(* PLC project Unnamed, Unknown Unnamed 1 *)
(* stored: creationDateTime 2025-10-10T14:27:24, modificationDateTime 2025-11-03T16:46:36 *)

PROGRAM rd_seq_rbear_trap
  VAR
    START : BOOL;
    PANIC : BOOL;
    Er : BOOL;
    SET_TRAP : BOOL;
    ACTIVATE_TRAP : BOOL;
    IN_MINUTOS : INT := 2;
    IN_SEGUNDOS : INT := 30;
    TIMER : INT;
    C_TIMER : INT;
    D_TIMER : INT;
    DISPLAY_M : INT;
    DISPLAY_S : INT;
    RANDOM : INT;
    RANDOM_ULINT : ULINT;
    SEED : ULINT := 0;
  END_VAR
  VAR CONSTANT
    M10 : ULINT := 10000;
    A : ULINT := 32310901;
    C : ULINT := 32310901;
    M : ULINT := 4294967296;
  END_VAR
  VAR
    Clock : BOOL;
    TOF0 : TOF;
    TON0 : TON;
    CTU_ULINT0 : CTU_ULINT;
    RESET : BOOL;
    D1 : INT;
    D2 : INT;
    D3 : INT;
    D4 : INT;
    CTU0 : CTU;
    R_TRIG1 : R_TRIG;
    CTU1 : CTU;
    TOF1 : TOF;
    CTU2 : CTU;
    TOF2 : TOF;
    CTU3 : CTU;
    TOF3 : TOF;
    CTU4 : CTU;
    TOF4 : TOF;
    B1 : BOOL;
    B2 : BOOL;
    B3 : BOOL;
    B4 : BOOL;
    M1 : BOOL;
    M2 : BOOL;
    M3 : BOOL;
    M4 : BOOL;
    E1 : BOOL;
    E2 : BOOL;
    E3 : BOOL;
    E4 : BOOL;
    R1 : BOOL;
    R2 : BOOL;
    R3 : BOOL;
    R4 : BOOL;
    G0 : BOOL;
    G1 : BOOL;
    G2 : BOOL;
    G3 : BOOL;
    G4 : BOOL;
    O1 : BOOL;
    O2 : BOOL;
    O3 : BOOL;
    O4 : BOOL;
    RELEASE_TRAP : BOOL;
    R_TRIG2 : R_TRIG;
    R_TRIG3 : R_TRIG;
    R_TRIG0 : R_TRIG;
    TON1 : TON;
  END_VAR
  VAR  (* added by the conversion: wires and edge detectors of the diagram *)
    R_TRIG1_2 : R_TRIG;
    R_TRIG2_2 : R_TRIG;
    _MUL1_ENO : BOOL;
    _MUL1_OUT : ULINT;
    _ADD5_ENO : BOOL;
    _ADD5_OUT : ULINT;
    _MOD7_ENO : BOOL;
    _MOD7_OUT : ULINT;
    R_TRIG3_2 : R_TRIG;
    R_TRIG4 : R_TRIG;
    R_TRIG5 : R_TRIG;
    R_TRIG6 : R_TRIG;
    _MUL17_ENO : BOOL;
    _MUL17_OUT : INT;
  END_VAR

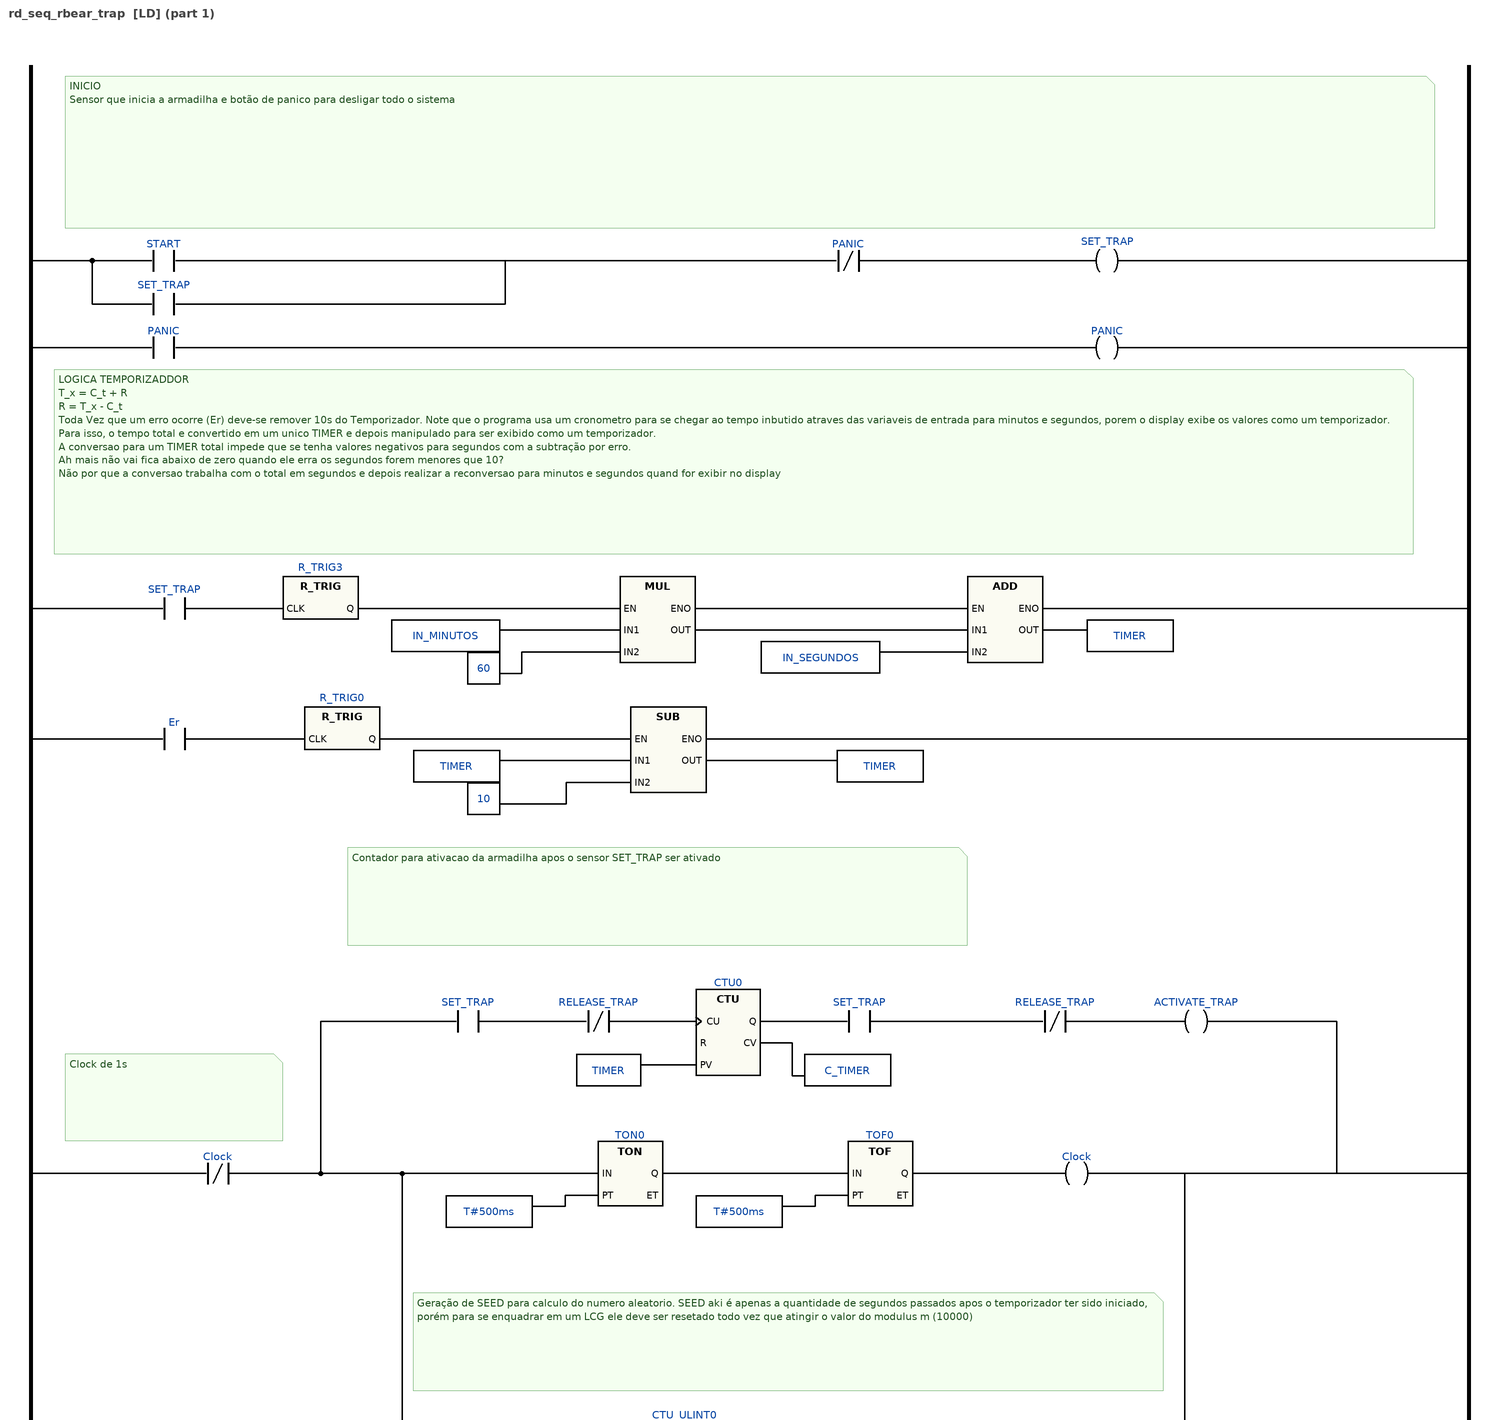
(* LD diagram, written out as Structured Text *)
(* INICIO
Sensor que inicia a armadilha e botão de panico para desligar todo o sistema *)
(* LOGICA TEMPORIZADDOR
T_x = C_t + R
R = T_x - C_t
Toda Vez que um erro ocorre (Er) deve-se remover 10s do Temporizador. Note que o programa usa um cronometro para se chegar ao tempo inbutido atraves das variaveis de entrada para minutos e segundos, porem o display exibe os valores como um temporizador. Para isso, o tempo total e convertido em um unico TIMER e depois manipulado para ser exibido como um temporizador.
A conversao para um TIMER total impede que se tenha valores negativos para segundos com a subtração por erro.
Ah mais não vai fica abaixo de zero quando ele erra os segundos forem menores que 10?
Não por que a conversao trabalha com o total em segundos e depois realizar a reconversao para minutos e segundos quand for exibir no display *)
(* Contador para ativacao da armadilha apos o sensor SET_TRAP ser ativado *)
(* Clock de 1s *)
TON0(IN := NOT Clock, PT := T#500ms);
TOF0(IN := TON0.Q, PT := T#500ms);
Clock := TOF0.Q;
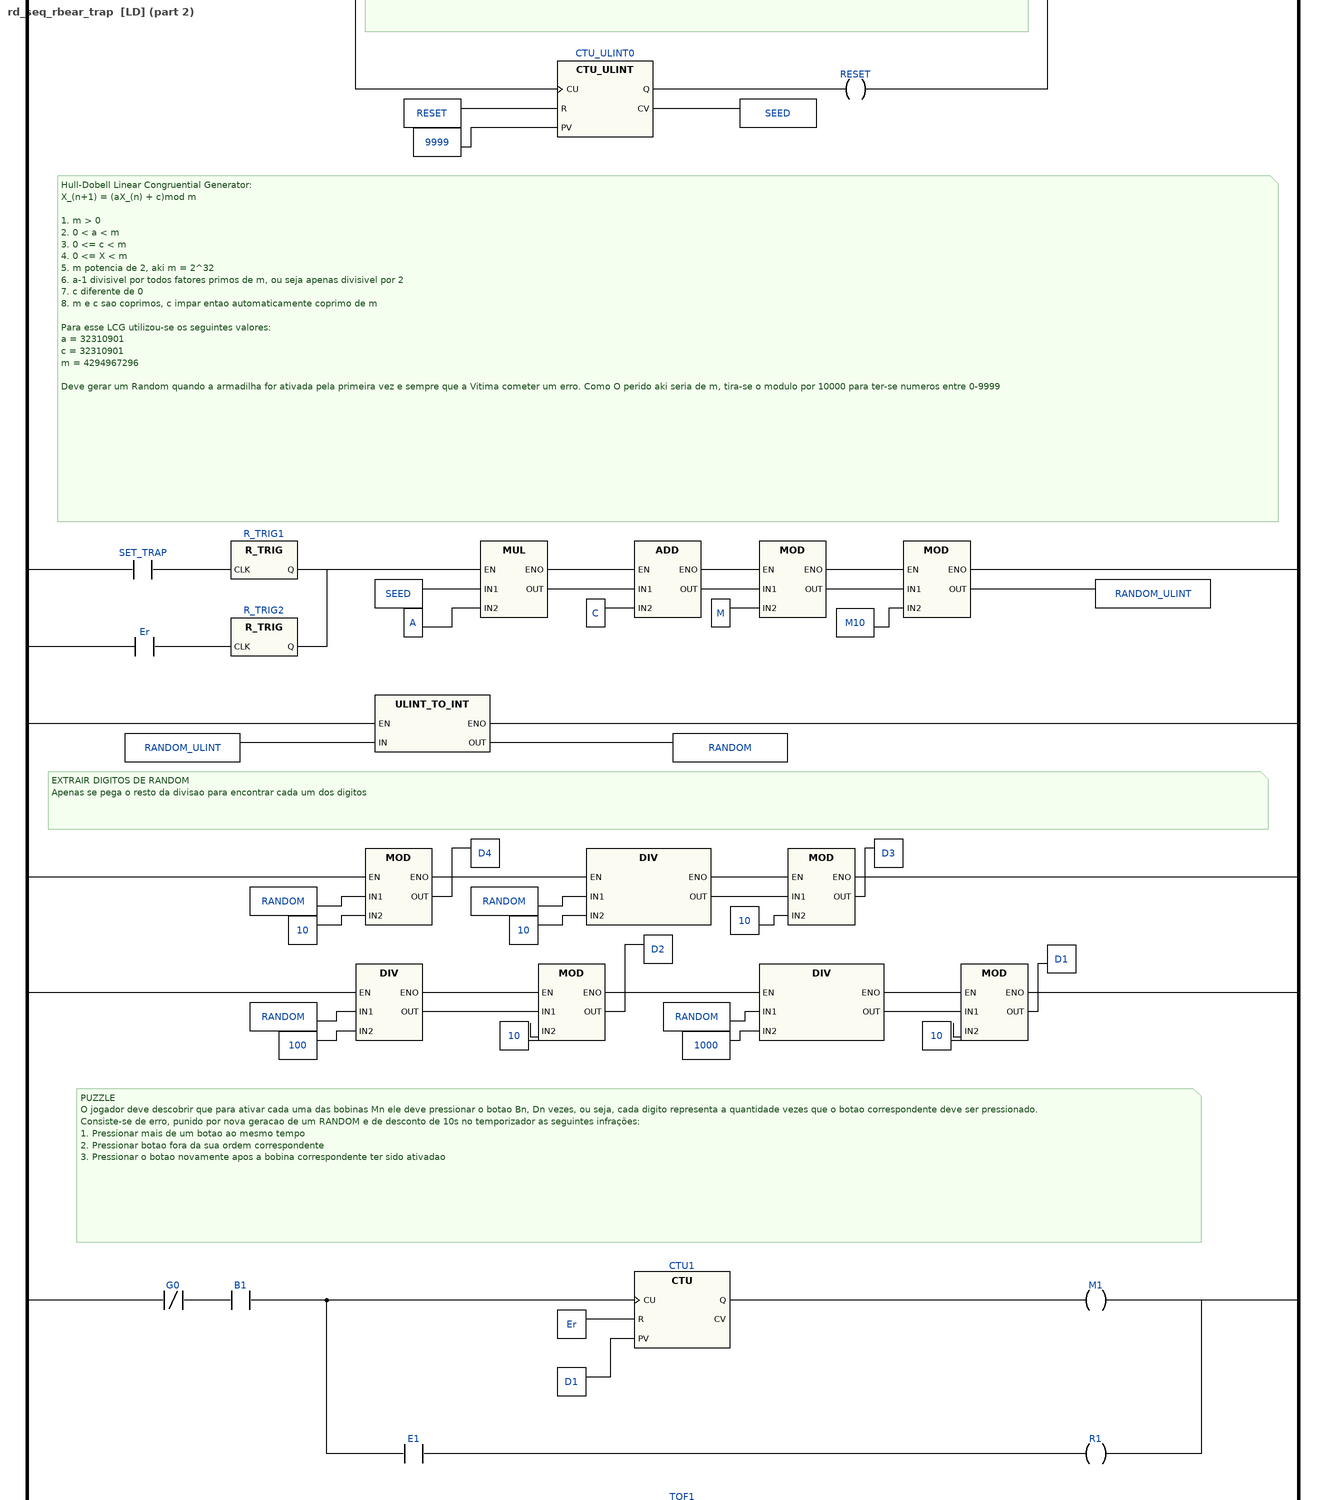
(* Geração de SEED para calculo do numero aleatorio. SEED aki é apenas a quantidade de segundos passados apos o temporizador ter sido iniciado, porém para se enquadrar em um LCG ele deve ser resetado todo vez que atingir o valor do modulus m (10000) *)
R_TRIG1_2(CLK := NOT Clock);
CTU_ULINT0(CU := R_TRIG1_2.Q, R := RESET, PV := 9999);
SEED := CTU_ULINT0.CV;
RESET := CTU_ULINT0.Q;
(* Hull-Dobell Linear Congruential Generator:
X_(n+1) = (aX_(n) + c)mod m

1. m > 0
2. 0 < a < m
3. 0 <= c < m
4. 0 <= X < m
5. m potencia de 2, aki m = 2^32
6. a-1 divisivel por todos fatores primos de m, ou seja apenas divisivel por 2
7. c diferente de 0
8. m e c sao coprimos, c impar entao automaticamente coprimo de m

Para esse LCG utilizou-se os seguintes valores:
   a = 32310901
   c = 32310901
   m = 4294967296

Deve gerar um Random quando a armadilha for ativada pela primeira vez e sempre que a Vitima cometer um erro. Como O perido aki seria de m, tira-se o modulo por 10000 para ter-se numeros entre 0-9999 *)
(* EXTRAIR DIGITOS DE RANDOM
Apenas se pega o resto da divisao para encontrar cada um dos digitos *)
D4 := RANDOM MOD 10;
D3 := RANDOM / 10 MOD 10;
D2 := RANDOM / 100 MOD 10;
D1 := RANDOM / 1000 MOD 10;
R_TRIG2_2(CLK := NOT Clock AND SET_TRAP AND NOT RELEASE_TRAP);
CTU0(CU := R_TRIG2_2.Q, PV := TIMER);
ACTIVATE_TRAP := CTU0.Q AND SET_TRAP AND NOT RELEASE_TRAP;
R_TRIG1(CLK := SET_TRAP);
R_TRIG2(CLK := Er);
_MUL1_OUT := MUL(EN := R_TRIG1.Q OR R_TRIG2.Q, IN1 := SEED, IN2 := A, ENO => _MUL1_ENO);
_ADD5_OUT := ADD(EN := _MUL1_ENO, IN1 := _MUL1_OUT, IN2 := C, ENO => _ADD5_ENO);
_MOD7_OUT := MOD(EN := _ADD5_ENO, IN1 := _ADD5_OUT, IN2 := M, ENO => _MOD7_ENO);
IF _MOD7_ENO THEN RANDOM_ULINT := _MOD7_OUT MOD M10; END_IF;
(* PUZZLE
O jogador deve descobrir que para ativar cada uma das bobinas Mn ele deve pressionar o botao Bn, Dn vezes, ou seja, cada digito representa a quantidade vezes que o botao correspondente deve ser pressionado.
Consiste-se de erro, punido por nova geracao de um RANDOM e de desconto de 10s no temporizador as seguintes infrações:
1. Pressionar mais de um botao ao mesmo tempo
2. Pressionar botao fora da sua ordem correspondente
3. Pressionar o botao novamente apos a bobina correspondente ter sido ativadao *)
R_TRIG3_2(CLK := NOT G0 AND B1);
CTU1(CU := R_TRIG3_2.Q, R := Er, PV := D1);
M1 := CTU1.Q;
R1 := NOT G0 AND B1 AND E1;
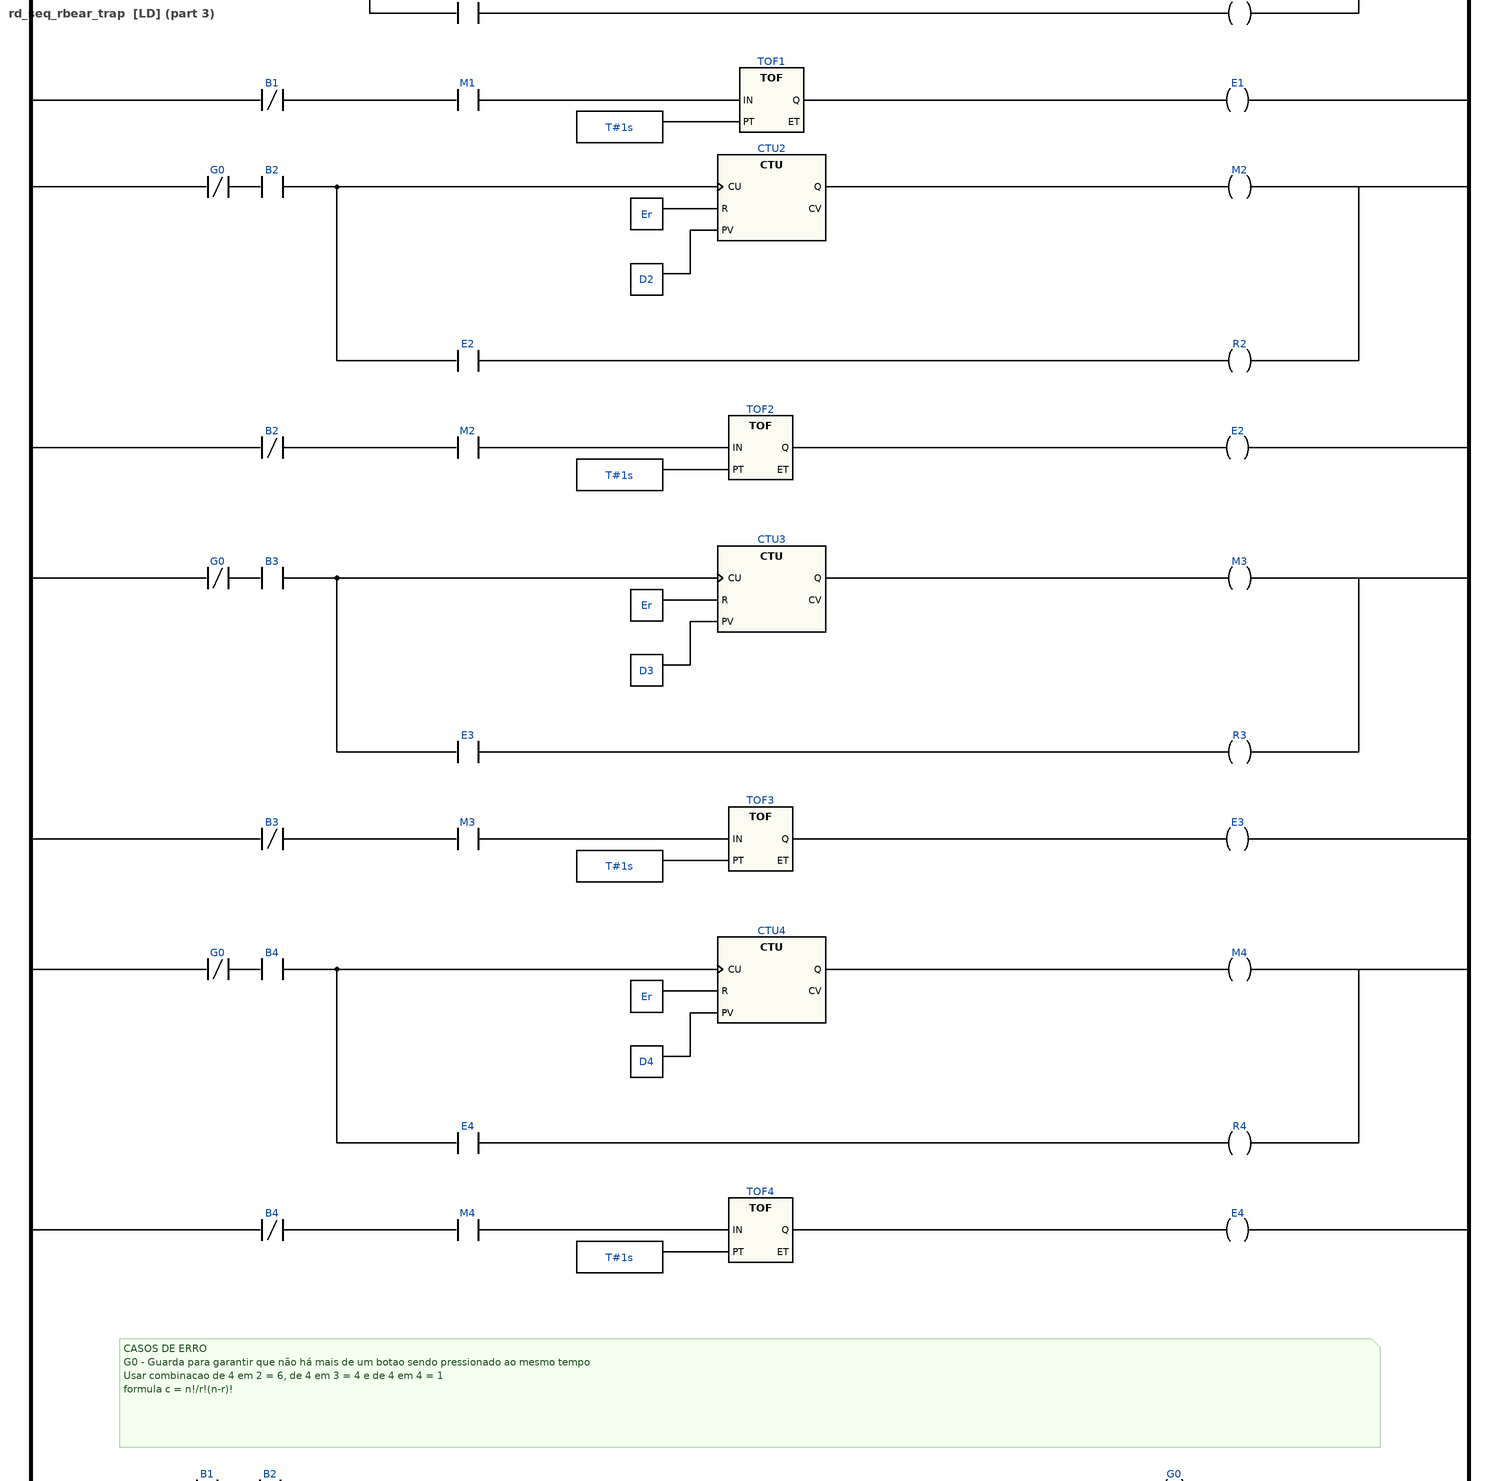
TOF1(IN := NOT B1 AND M1, PT := T#1s);
E1 := TOF1.Q;
R_TRIG4(CLK := NOT G0 AND B2);
CTU2(CU := R_TRIG4.Q, R := Er, PV := D2);
M2 := CTU2.Q;
R2 := NOT G0 AND B2 AND E2;
TOF2(IN := NOT B2 AND M2, PT := T#1s);
E2 := TOF2.Q;
R_TRIG5(CLK := NOT G0 AND B3);
CTU3(CU := R_TRIG5.Q, R := Er, PV := D3);
M3 := CTU3.Q;
R3 := NOT G0 AND B3 AND E3;
TOF3(IN := NOT B3 AND M3, PT := T#1s);
E3 := TOF3.Q;
R_TRIG6(CLK := NOT G0 AND B4);
CTU4(CU := R_TRIG6.Q, R := Er, PV := D4);
M4 := CTU4.Q;
R4 := NOT G0 AND B4 AND E4;
TOF4(IN := NOT B4 AND M4, PT := T#1s);
E4 := TOF4.Q;
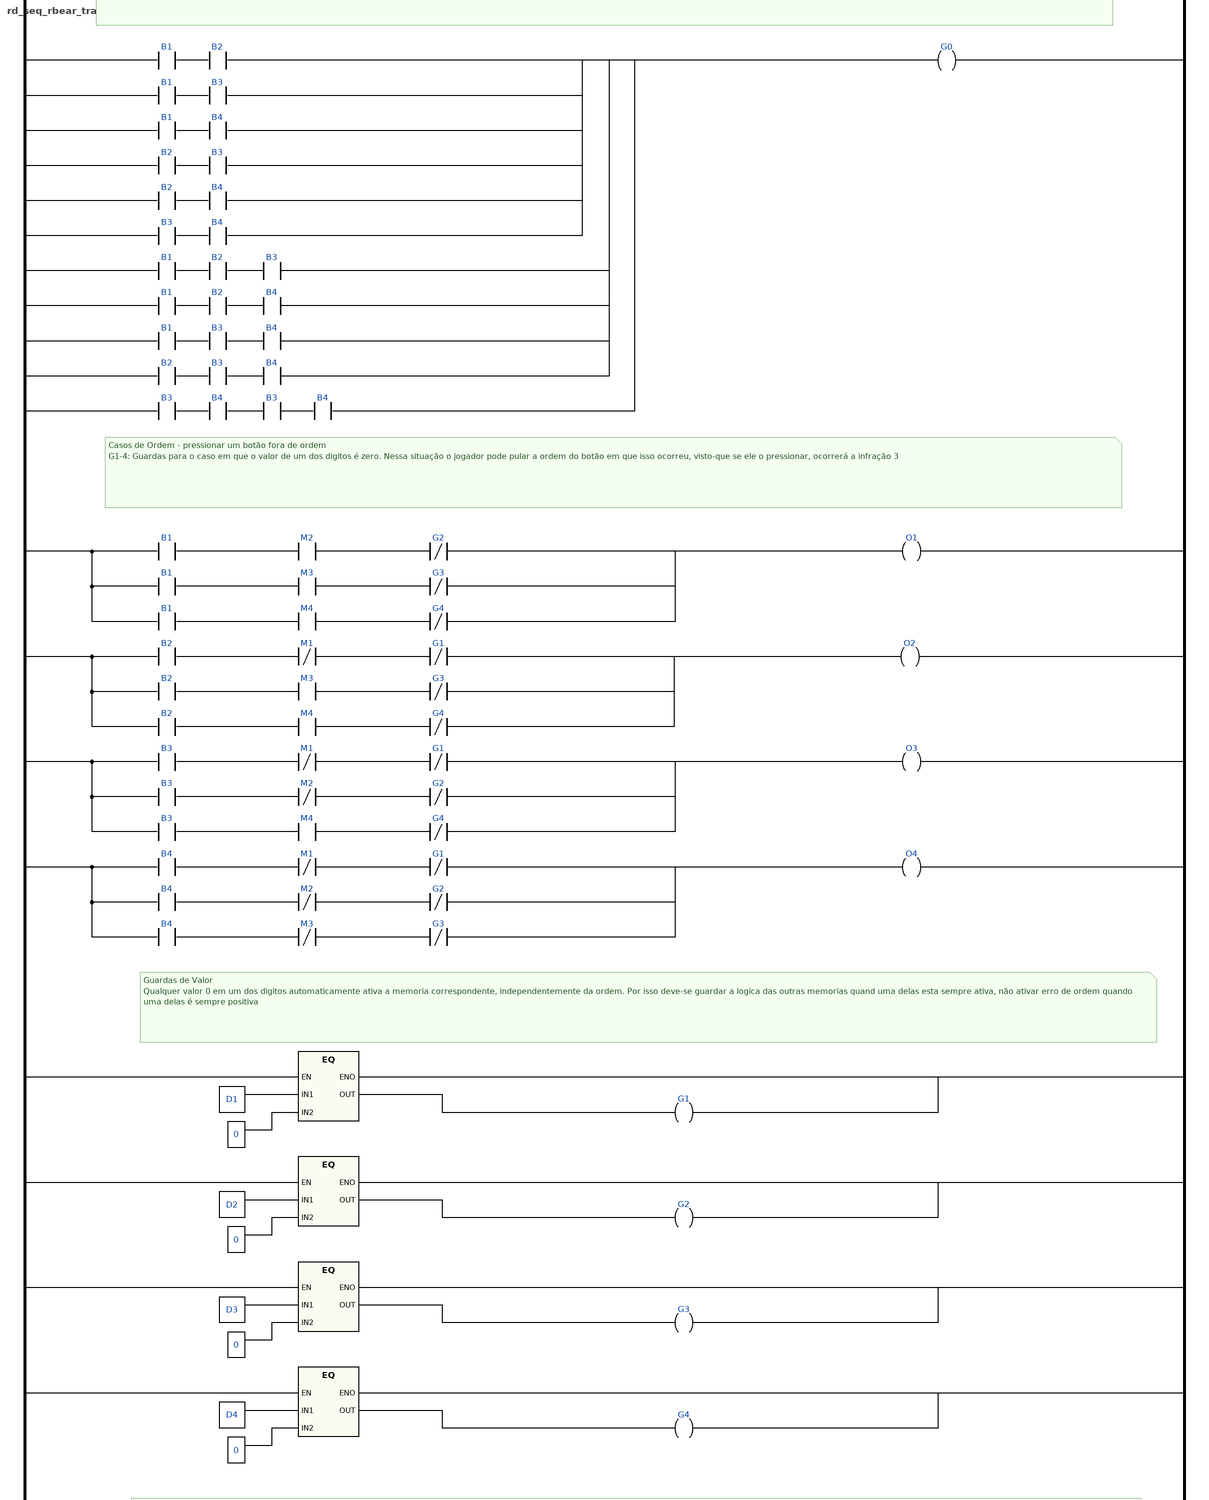
(* CASOS DE ERRO
G0 - Guarda para garantir que não há mais de um botao sendo pressionado ao mesmo tempo
Usar combinacao de 4 em 2 = 6, de 4 em 3 = 4 e de 4 em 4 = 1 
formula c = n!/r!(n-r)! *)
G0 := B1 AND B2 OR B1 AND B3 OR B1 AND B4 OR B2 AND B3 OR B2 AND B4 OR B3 AND B4 OR B1 AND B2 AND B3 OR B1 AND B2 AND B4 OR B1 AND B3 AND B4 OR B2 AND B3 AND B4 OR B3 AND B4 AND B3 AND B4;
(* Casos de Ordem - pressionar um botão fora de ordem
G1-4: Guardas para o caso em que o valor de um dos digitos é zero. Nessa situação o jogador pode pular a ordem do botão em que isso ocorreu, visto-que se ele o pressionar, ocorrerá a infração 3 *)
O1 := B1 AND (M2 AND NOT G2 OR M3 AND NOT G3 OR M4 AND NOT G4);
O2 := B2 AND (NOT M1 AND NOT G1 OR M3 AND NOT G3 OR M4 AND NOT G4);
O3 := B3 AND (NOT M1 AND NOT G1 OR NOT M2 AND NOT G2 OR M4 AND NOT G4);
O4 := B4 AND (NOT M1 AND NOT G1 OR NOT M2 AND NOT G2 OR NOT M3 AND NOT G3);
(* Guardas de Valor
Qualquer valor 0 em um dos digitos automaticamente ativa a memoria correspondente, independentemente da ordem. Por isso deve-se guardar a logica das outras memorias quand uma delas esta sempre ativa, não ativar erro de ordem quando uma delas é sempre positiva *)
G1 := D1 = 0;
G2 := D2 = 0;
G3 := D3 = 0;
G4 := D4 = 0;
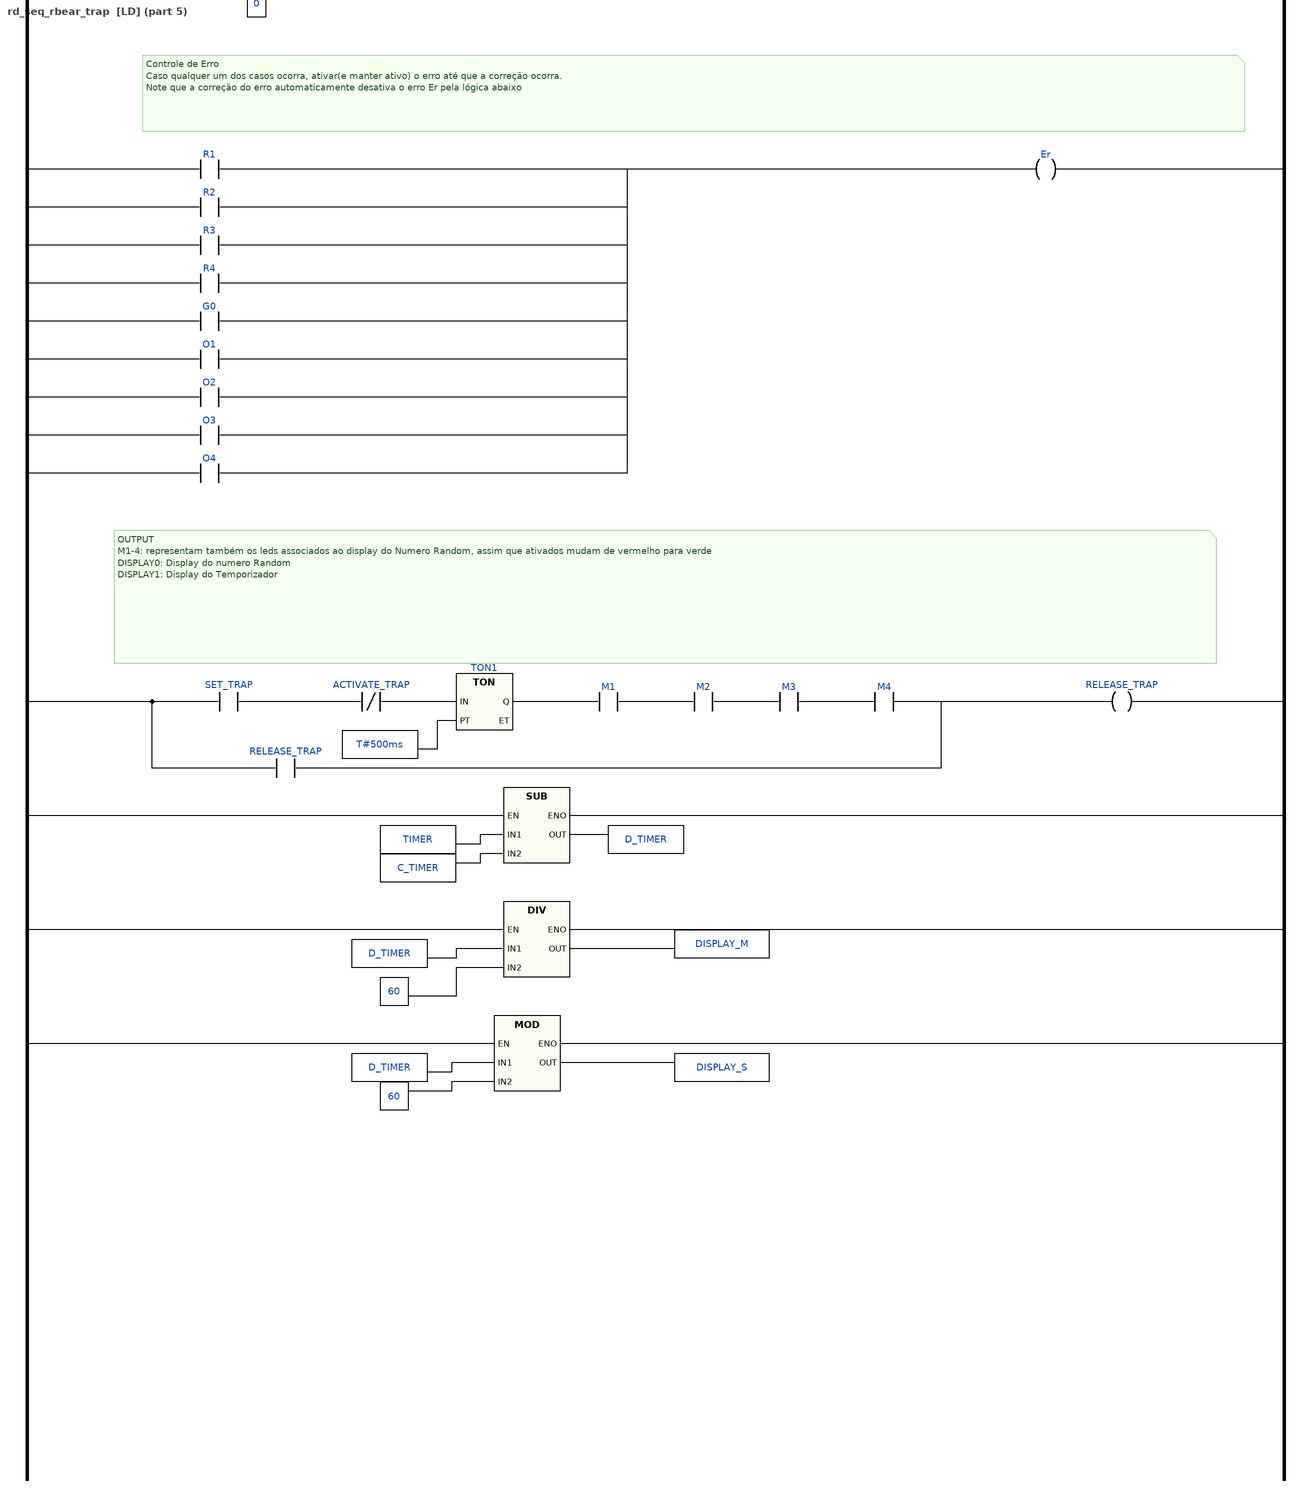
(* Controle de Erro
Caso qualquer um dos casos ocorra, ativar(e manter ativo) o erro até que a correção ocorra.
Note que a correção do erro automaticamente desativa o erro Er pela lógica abaixo *)
Er := R1 OR R2 OR R3 OR R4 OR G0 OR O1 OR O2 OR O3 OR O4;
(* OUTPUT
M1-4: representam também os leds associados ao display do Numero Random, assim que ativados mudam de vermelho para verde
DISPLAY0: Display do numero Random
DISPLAY1: Display do Temporizador *)
TON1(IN := SET_TRAP AND NOT ACTIVATE_TRAP, PT := T#500ms);
RELEASE_TRAP := TON1.Q AND M1 AND M2 AND M3 AND M4 OR RELEASE_TRAP;
RANDOM := ULINT_TO_INT(RANDOM_ULINT);
SET_TRAP := (START OR SET_TRAP) AND NOT PANIC;
PANIC := PANIC;
R_TRIG3(CLK := SET_TRAP);
_MUL17_OUT := MUL(EN := R_TRIG3.Q, IN1 := IN_MINUTOS, IN2 := 60, ENO => _MUL17_ENO);
IF _MUL17_ENO THEN TIMER := _MUL17_OUT + IN_SEGUNDOS; END_IF;
R_TRIG0(CLK := Er);
IF R_TRIG0.Q THEN TIMER := TIMER - 10; END_IF;
C_TIMER := CTU0.CV;
DISPLAY_S := D_TIMER MOD 60;
DISPLAY_M := D_TIMER / 60;
D_TIMER := TIMER - C_TIMER;
END_PROGRAM

PROGRAM my_clock_counter
  VAR
    Clock : BOOL;
    Clock0 : BOOL;
    DISPLAY : ULINT;
    TON0 : TON;
    TOF0 : TOF;
    CTU_ULINT0 : CTU_ULINT;
    Reset : BOOL;
  END_VAR
  VAR  (* added by the conversion: wires and edge detectors of the diagram *)
    R_TRIG1 : R_TRIG;
  END_VAR

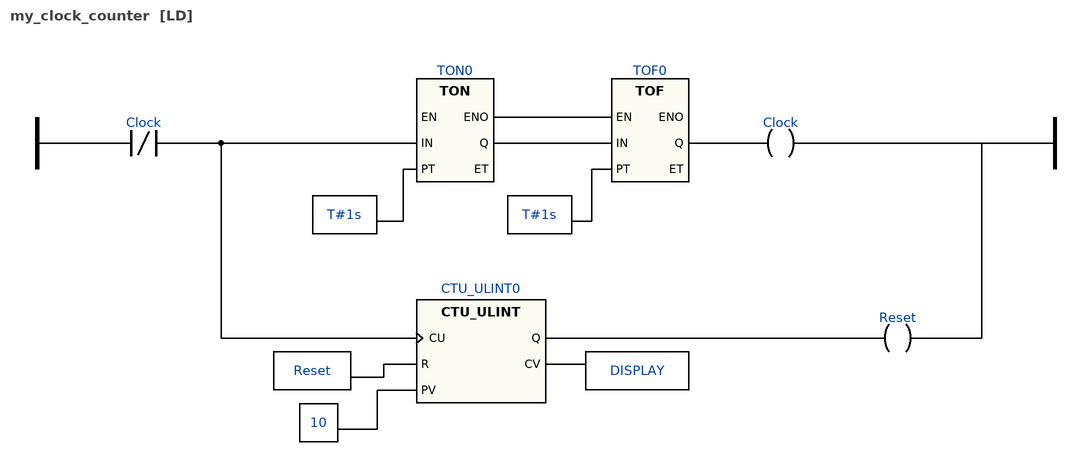
(* LD diagram, written out as Structured Text *)
TON0(IN := NOT Clock, PT := T#1s);
TOF0(EN := TON0.ENO, IN := TON0.Q, PT := T#1s);
Clock := TOF0.Q;
R_TRIG1(CLK := NOT Clock);
CTU_ULINT0(CU := R_TRIG1.Q, R := Reset, PV := 10);
DISPLAY := CTU_ULINT0.CV;
Reset := CTU_ULINT0.Q;
END_PROGRAM

PROGRAM digit_extractor
  VAR
    RANDOM : ULINT := 1234;
    DIVISOR : ULINT := 10;
  END_VAR
  VAR RETAIN
    D1 : ULINT;
  END_VAR
  VAR
    D2 : ULINT;
    D3 : ULINT;
    D4 : ULINT;
    M1 : BOOL;
  END_VAR

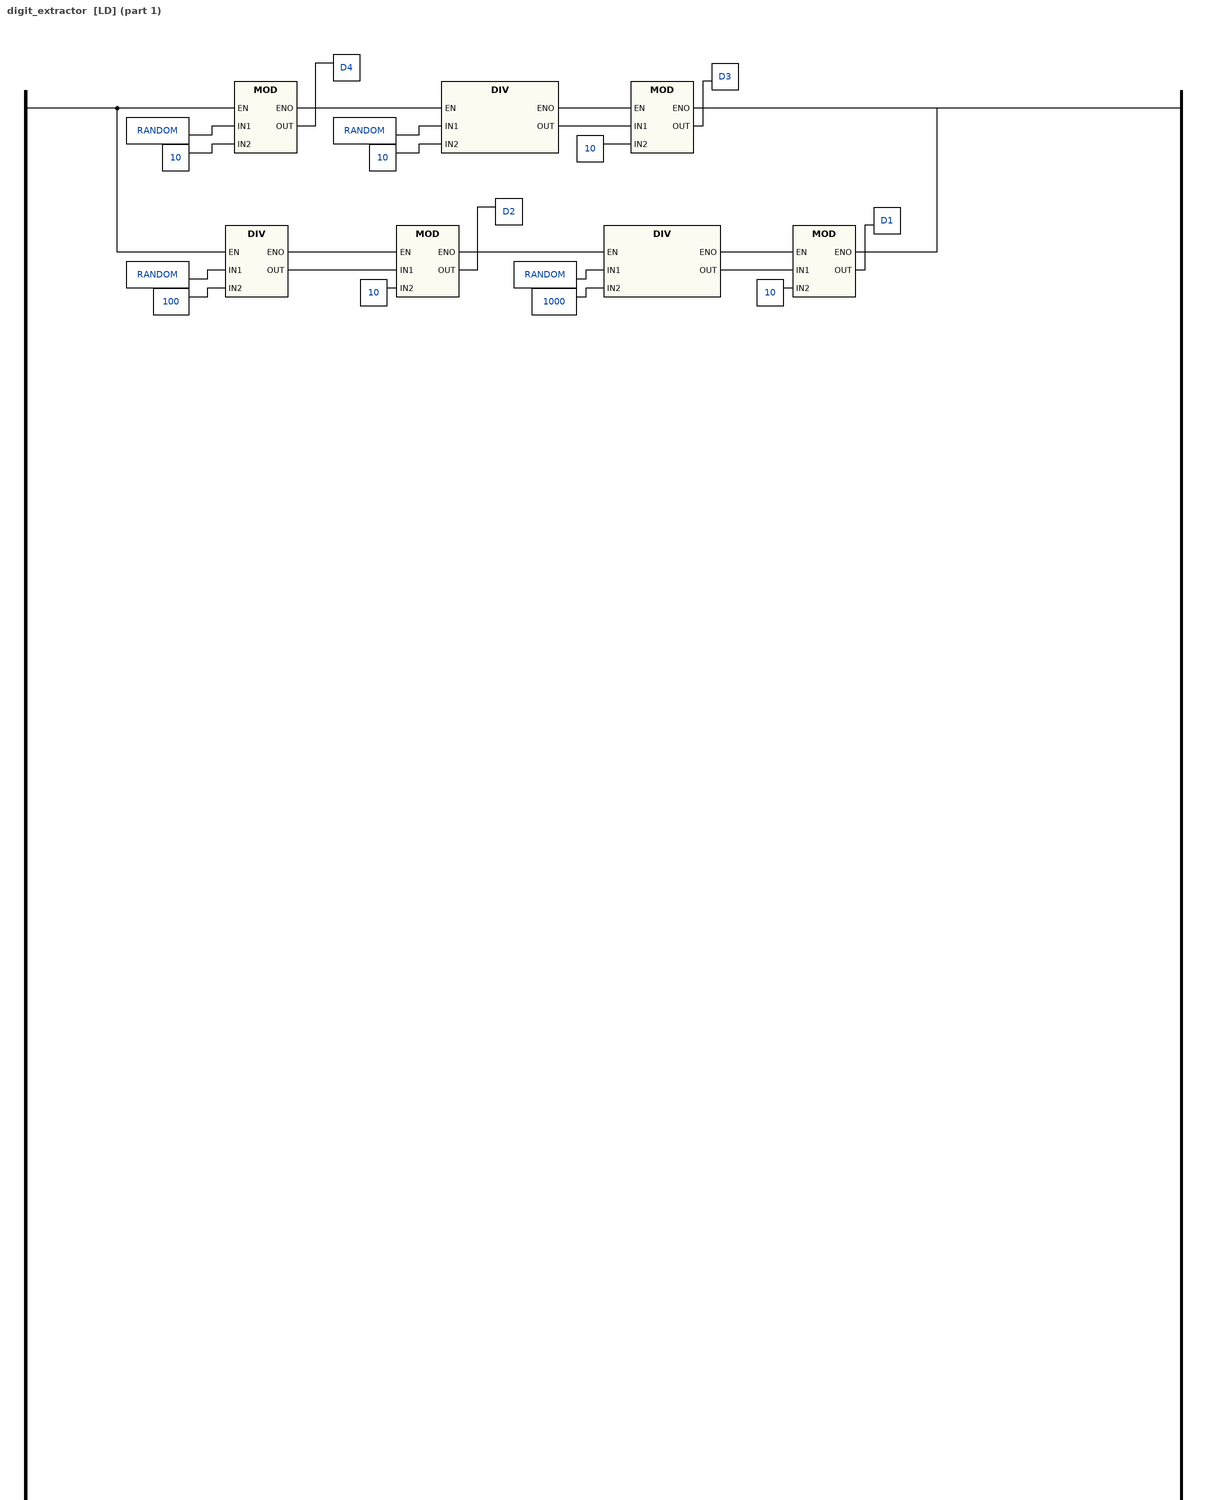
(* LD diagram, written out as Structured Text *)
D4 := RANDOM MOD 10;
D3 := RANDOM / 10 MOD 10;
D2 := RANDOM / 100 MOD 10;
D1 := RANDOM / 1000 MOD 10;
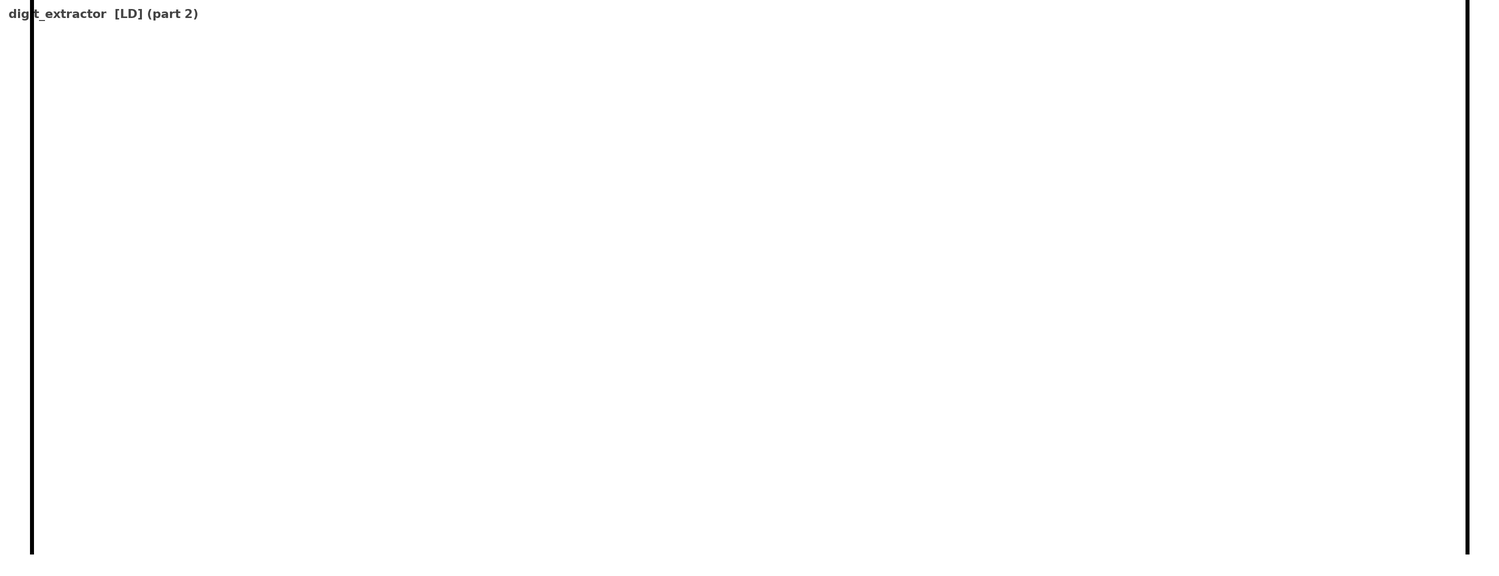
END_PROGRAM

PROGRAM puzzle
  VAR
    D1 : INT := 1;
    D2 : INT := 1;
    D3 : INT := 1;
    D4 : INT := 1;
    B1 : BOOL;
    B2 : BOOL;
    B3 : BOOL;
    B4 : BOOL;
    M1 : BOOL;
    M2 : BOOL;
    M3 : BOOL;
    M4 : BOOL;
    E1 : BOOL;
    E2 : BOOL;
    E3 : BOOL;
    E4 : BOOL;
    CTU1 : CTU;
    R1 : BOOL;
    R2 : BOOL;
    R3 : BOOL;
    R4 : BOOL;
    G1 : BOOL;
    G2 : BOOL;
    G3 : BOOL;
    G4 : BOOL;
    G0 : BOOL;
    O1 : BOOL;
    O2 : BOOL;
    O3 : BOOL;
    O4 : BOOL;
    Er : BOOL;
    SAFE : BOOL;
    CTU2 : CTU;
    CTU3 : CTU;
    CTU4 : CTU;
  END_VAR
  VAR  (* added by the conversion: wires and edge detectors of the diagram *)
    R_TRIG1 : R_TRIG;
    R_TRIG2 : R_TRIG;
    R_TRIG3 : R_TRIG;
    R_TRIG4 : R_TRIG;
  END_VAR

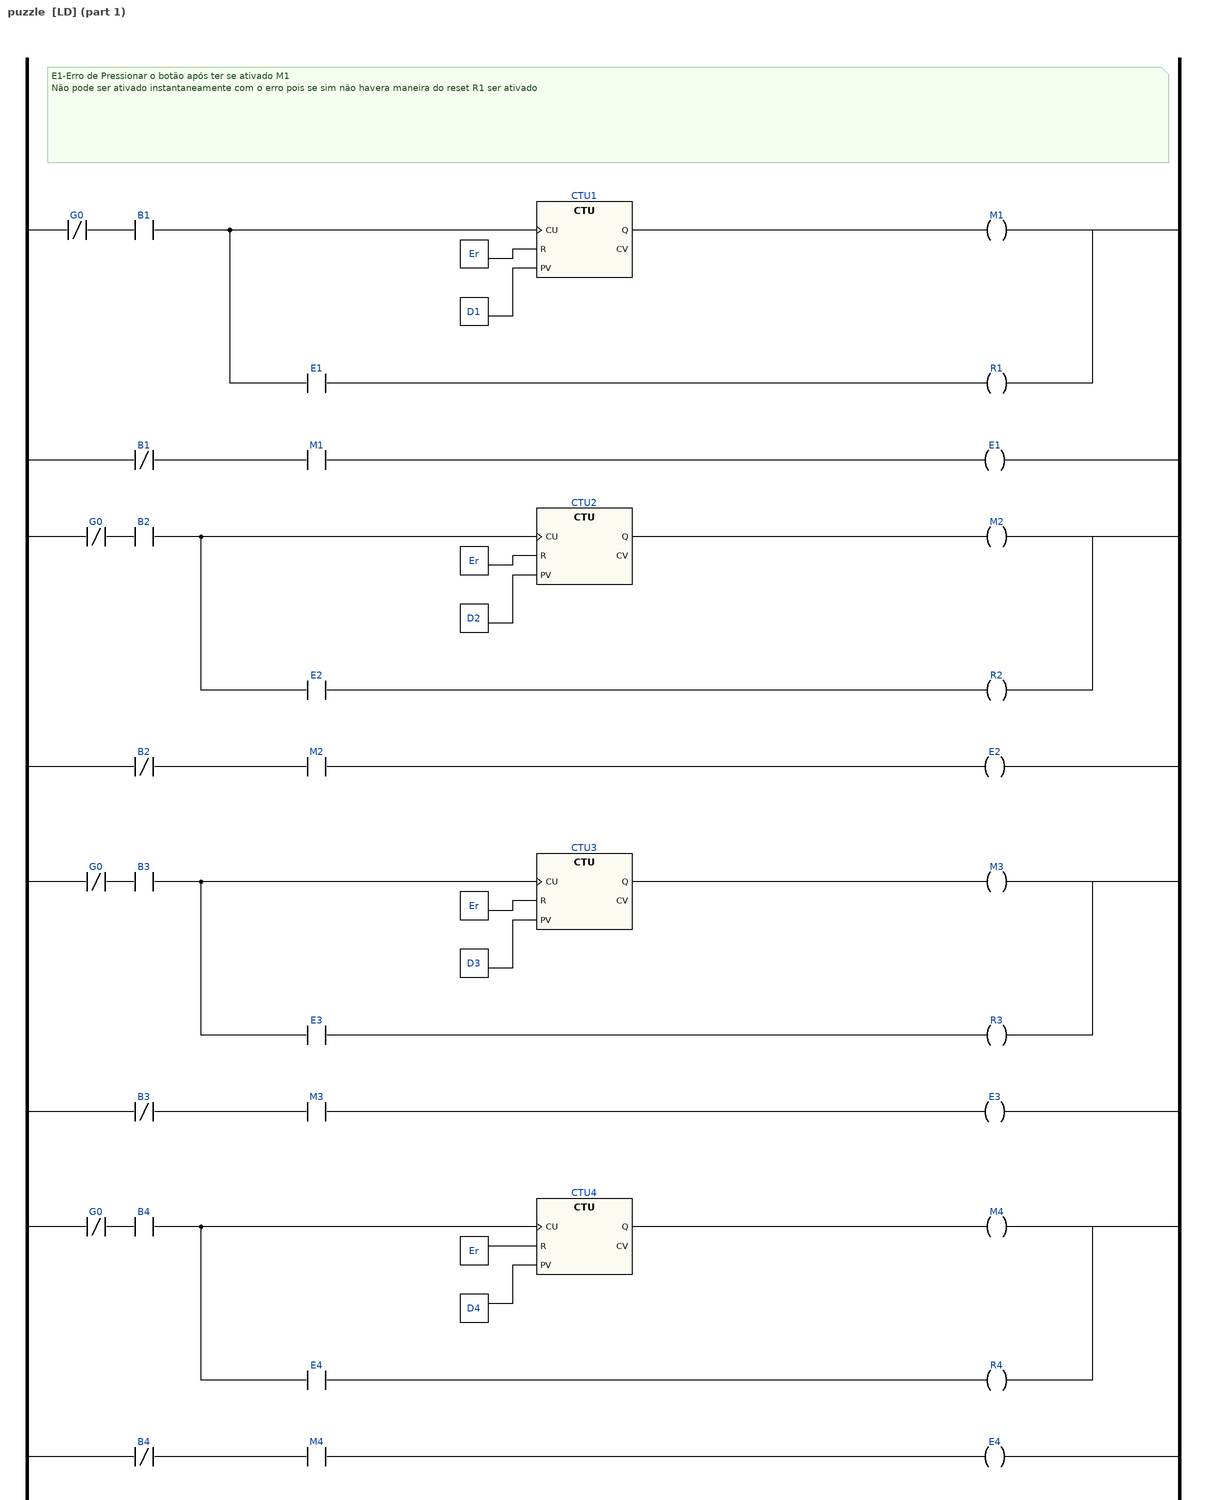
(* LD diagram, written out as Structured Text *)
(* E1-Erro de Pressionar o botão após ter se ativado M1
Não pode ser ativado instantaneamente com o erro pois se sim não havera maneira do reset R1 ser ativado *)
R_TRIG1(CLK := NOT G0 AND B1);
CTU1(CU := R_TRIG1.Q, R := Er, PV := D1);
M1 := CTU1.Q;
R1 := NOT G0 AND B1 AND E1;
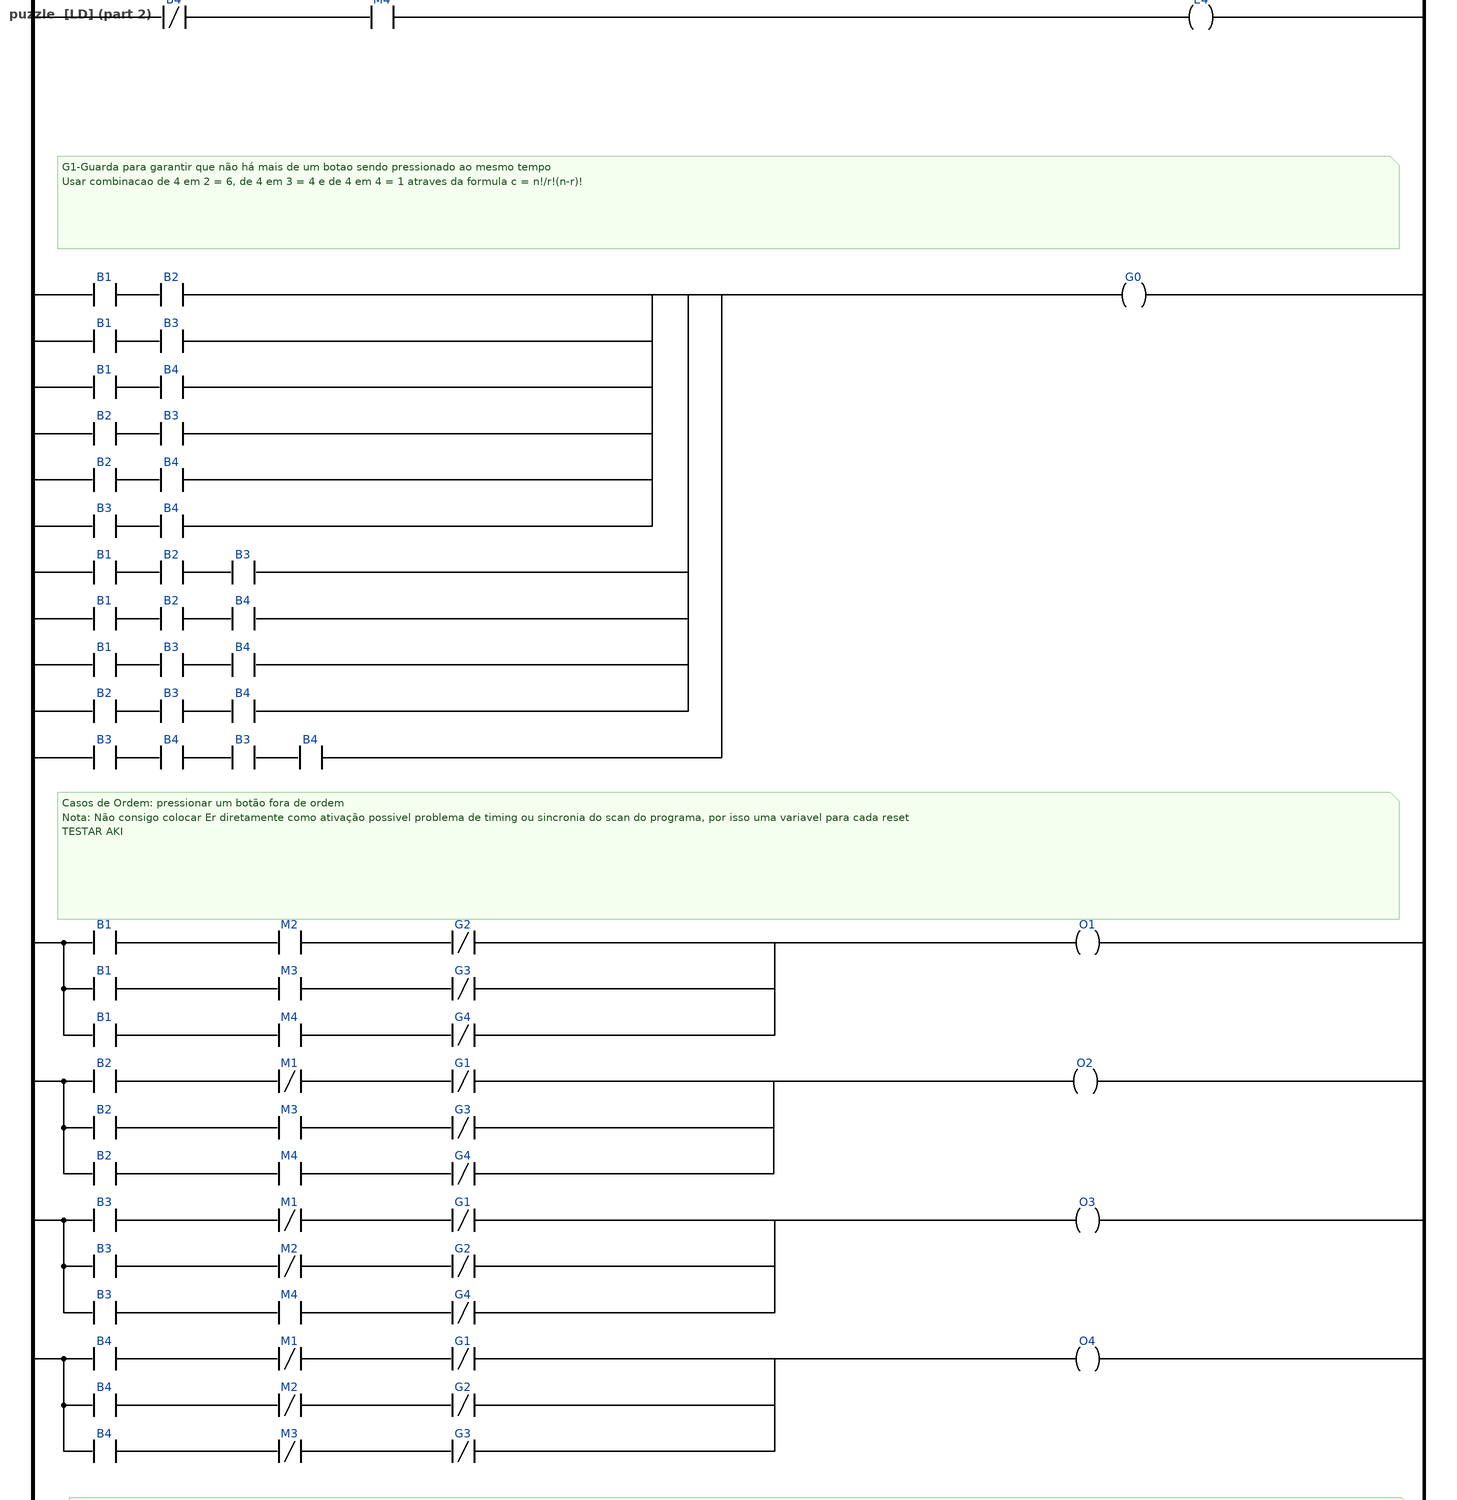
(* G1-Guarda para garantir que não há mais de um botao sendo pressionado ao mesmo tempo
Usar combinacao de 4 em 2 = 6, de 4 em 3 = 4 e de 4 em 4 = 1 atraves da formula c = n!/r!(n-r)! *)
G0 := B1 AND B2 OR B1 AND B3 OR B1 AND B4 OR B2 AND B3 OR B2 AND B4 OR B3 AND B4 OR B1 AND B2 AND B3 OR B1 AND B2 AND B4 OR B1 AND B3 AND B4 OR B2 AND B3 AND B4 OR B3 AND B4 AND B3 AND B4;
(* Casos de Ordem: pressionar um botão fora de ordem
Nota: Não consigo colocar Er diretamente como ativação possivel problema de timing ou sincronia do scan do programa, por isso uma variavel para cada reset
TESTAR AKI *)
O1 := B1 AND (M2 AND NOT G2 OR M3 AND NOT G3 OR M4 AND NOT G4);
R_TRIG2(CLK := NOT G0 AND B2);
CTU2(CU := R_TRIG2.Q, R := Er, PV := D2);
M2 := CTU2.Q;
R2 := NOT G0 AND B2 AND E2;
E2 := NOT B2 AND M2;
R_TRIG3(CLK := NOT G0 AND B3);
CTU3(CU := R_TRIG3.Q, R := Er, PV := D3);
M3 := CTU3.Q;
R3 := NOT G0 AND B3 AND E3;
E3 := NOT B3 AND M3;
R_TRIG4(CLK := NOT G0 AND B4);
CTU4(CU := R_TRIG4.Q, R := Er, PV := D4);
M4 := CTU4.Q;
R4 := NOT G0 AND B4 AND E4;
E4 := NOT B4 AND M4;
O2 := B2 AND (NOT M1 AND NOT G1 OR M3 AND NOT G3 OR M4 AND NOT G4);
O3 := B3 AND (NOT M1 AND NOT G1 OR NOT M2 AND NOT G2 OR M4 AND NOT G4);
O4 := B4 AND (NOT M1 AND NOT G1 OR NOT M2 AND NOT G2 OR NOT M3 AND NOT G3);
E1 := NOT B1 AND M1;
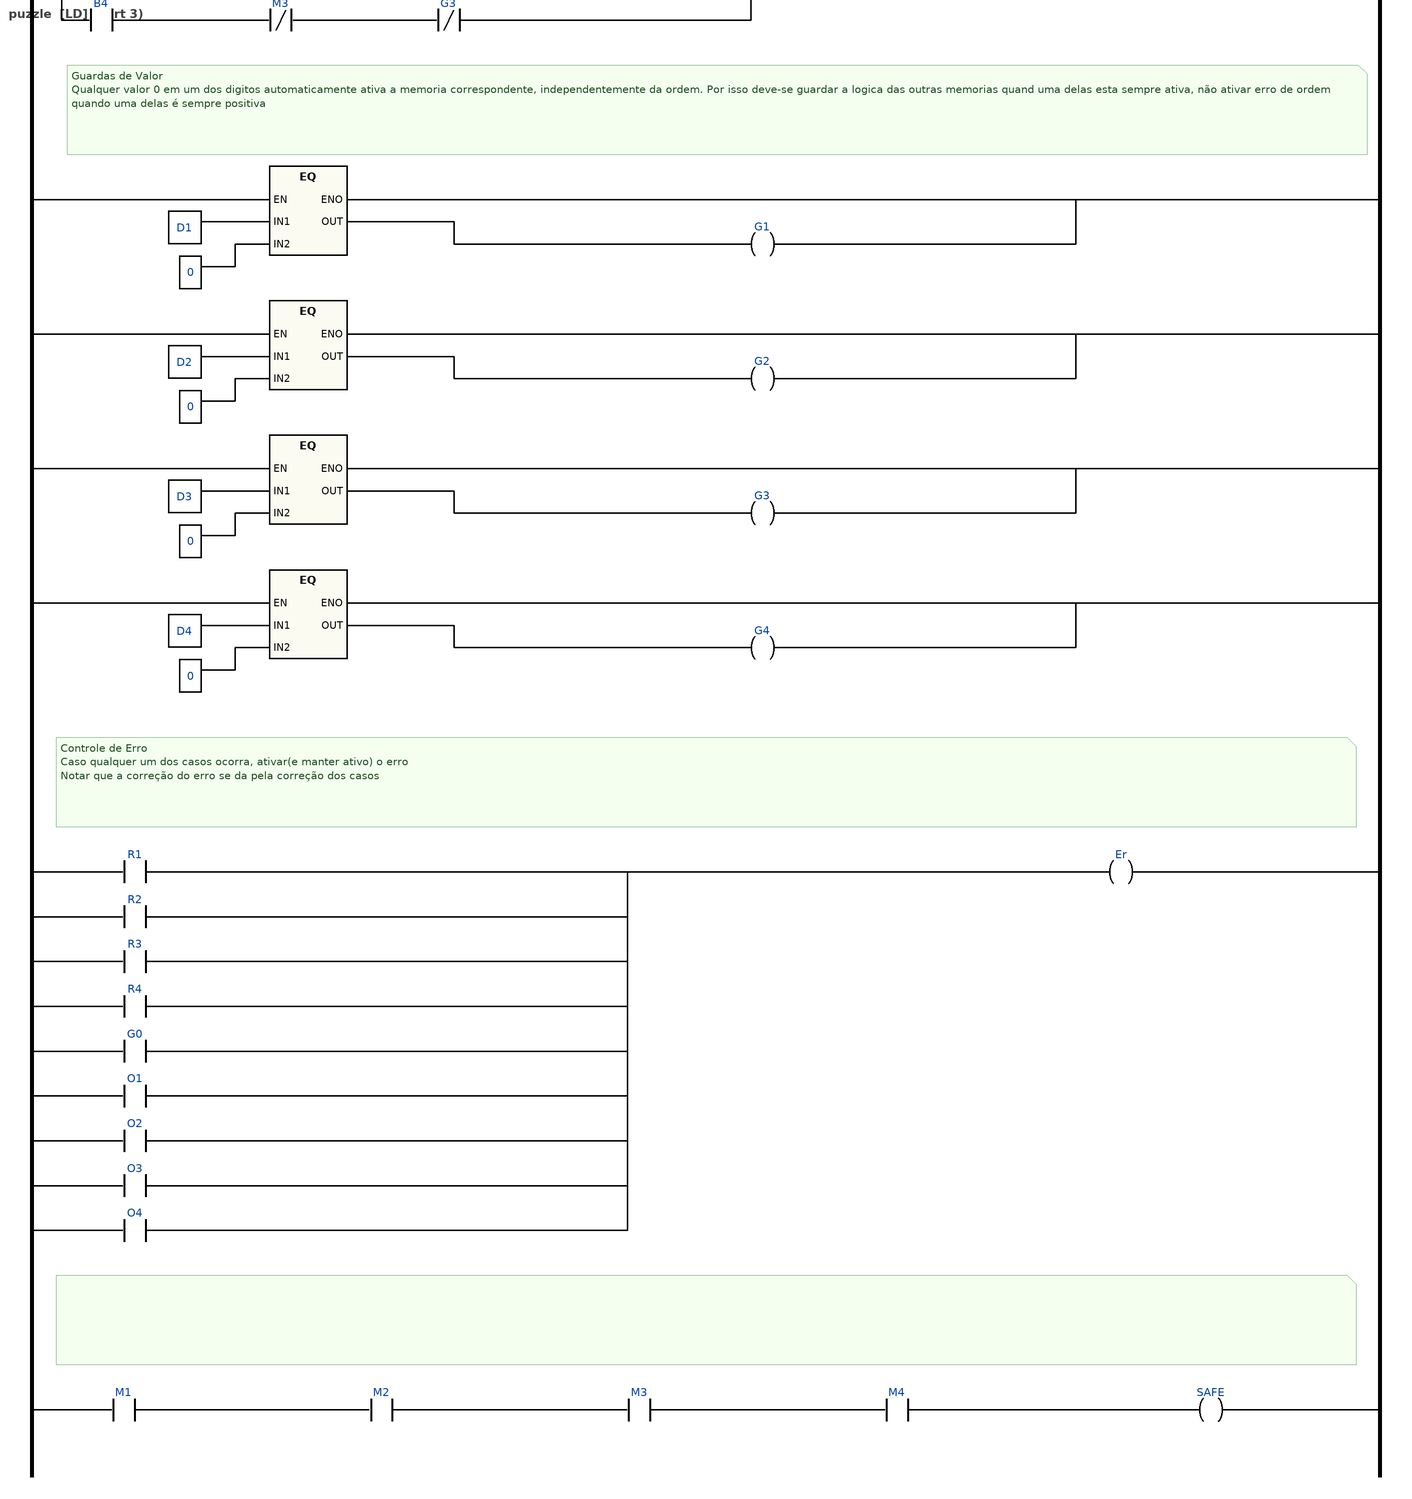
(* Guardas de Valor
Qualquer valor 0 em um dos digitos automaticamente ativa a memoria correspondente, independentemente da ordem. Por isso deve-se guardar a logica das outras memorias quand uma delas esta sempre ativa, não ativar erro de ordem quando uma delas é sempre positiva *)
G1 := D1 = 0;
G2 := D2 = 0;
G3 := D3 = 0;
G4 := D4 = 0;
(* Controle de Erro
Caso qualquer um dos casos ocorra, ativar(e manter ativo) o erro
Notar que a correção do erro se da pela correção dos casos *)
Er := R1 OR R2 OR R3 OR R4 OR G0 OR O1 OR O2 OR O3 OR O4;
SAFE := M1 AND M2 AND M3 AND M4;
END_PROGRAM

PROGRAM sub_timer
  VAR
    Er : BOOL;
    START : BOOL;
    PANIC : BOOL;
    IN_MINUTOS : INT := 2;
    IN_SEGUNDOS : INT := 20;
    R_SEGUNDOS : BOOL;
    DISPLAY_M : INT;
    DISPLAY_S : INT;
    Clock : BOOL;
    I_TIMER : INT;
    TIMER : INT;
    C_TIMER : INT;
    D_TIMER : INT;
    TOF0 : TOF;
    TON0 : TON;
    SET_TRAP : BOOL;
    ACTIVATE_TRAP : BOOL;
    CTU0 : CTU;
    R_TRIG0 : R_TRIG;
    R_TRIG1 : R_TRIG;
  END_VAR
  VAR  (* added by the conversion: wires and edge detectors of the diagram *)
    R_TRIG1_2 : R_TRIG;
    _MUL86_ENO : BOOL;
    _MUL86_OUT : INT;
  END_VAR

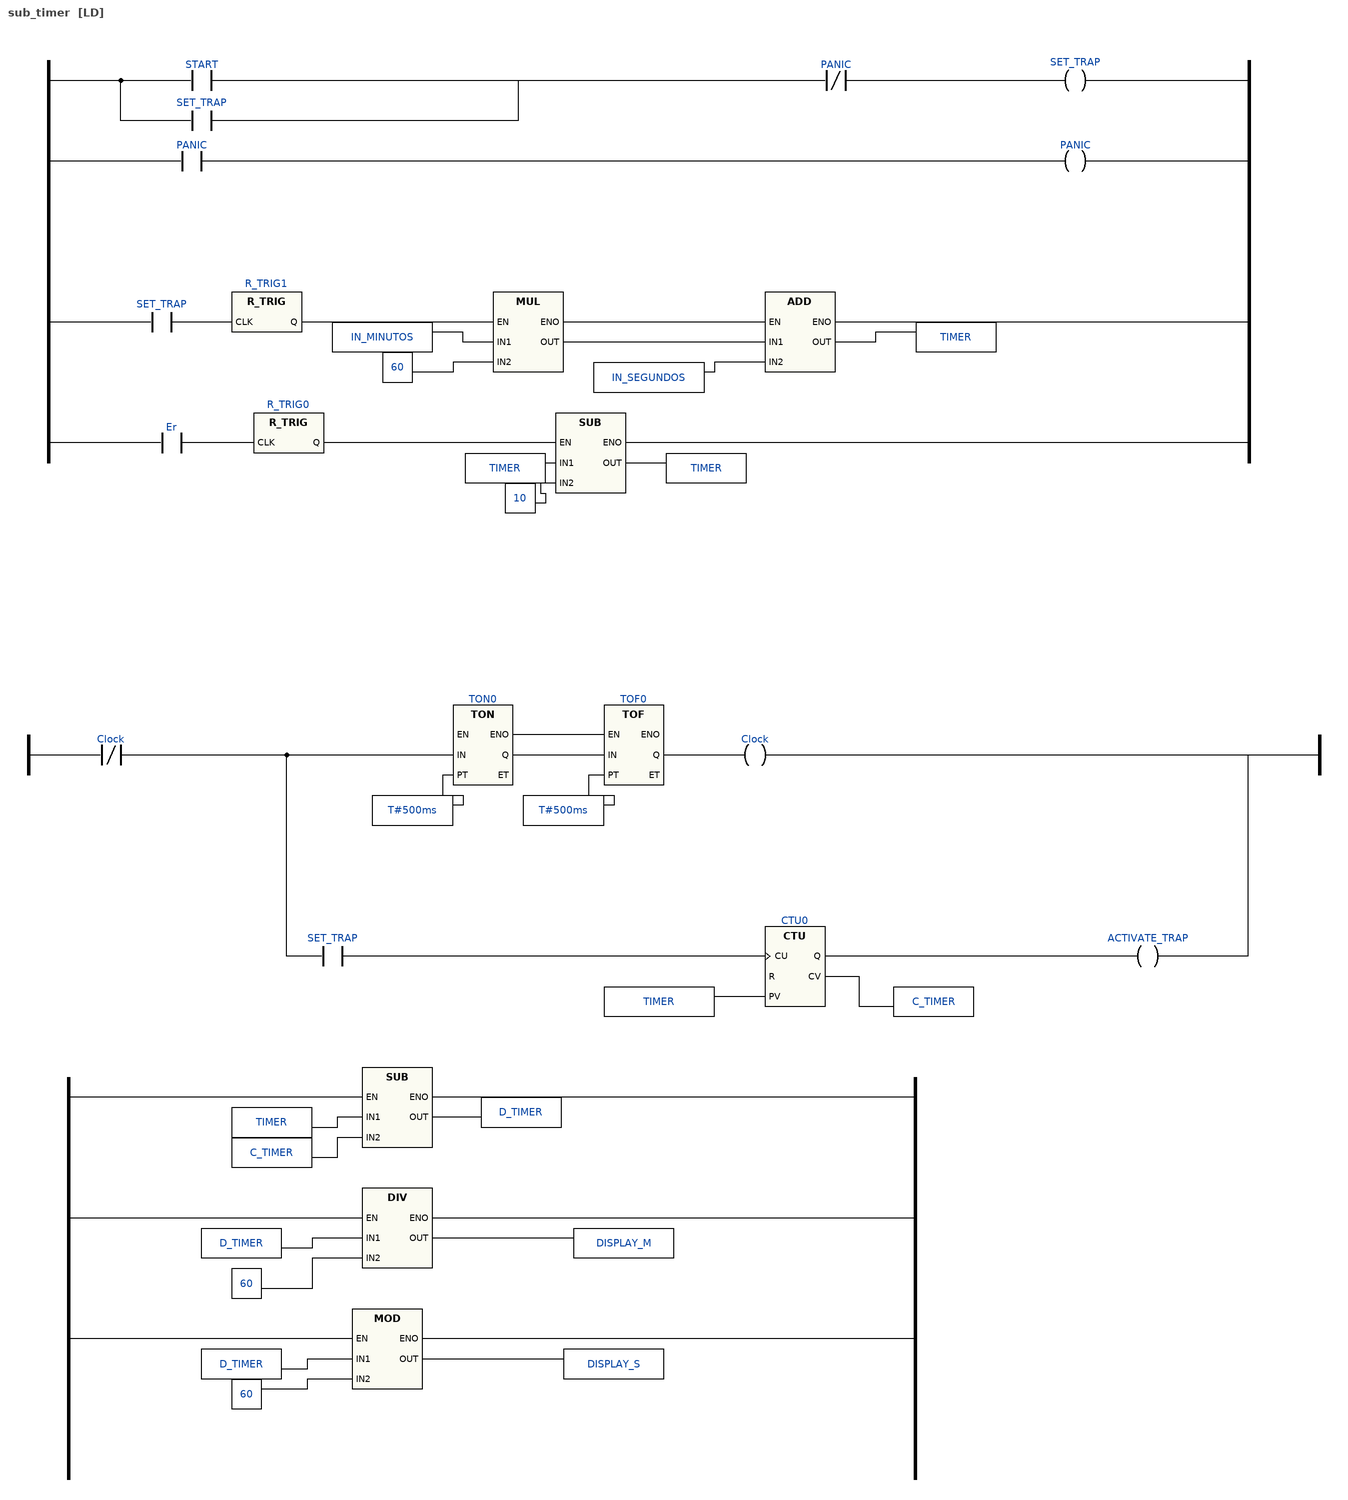
(* LD diagram, written out as Structured Text *)
TON0(IN := NOT Clock, PT := T#500ms);
TOF0(EN := TON0.ENO, IN := TON0.Q, PT := T#500ms);
Clock := TOF0.Q;
R_TRIG1_2(CLK := NOT Clock AND SET_TRAP);
CTU0(CU := R_TRIG1_2.Q, PV := TIMER);
ACTIVATE_TRAP := CTU0.Q;
SET_TRAP := (START OR SET_TRAP) AND NOT PANIC;
DISPLAY_S := D_TIMER MOD 60;
DISPLAY_M := D_TIMER / 60;
R_TRIG1(CLK := SET_TRAP);
_MUL86_OUT := MUL(EN := R_TRIG1.Q, IN1 := IN_MINUTOS, IN2 := 60, ENO => _MUL86_ENO);
IF _MUL86_ENO THEN TIMER := _MUL86_OUT + IN_SEGUNDOS; END_IF;
C_TIMER := CTU0.CV;
D_TIMER := TIMER - C_TIMER;
R_TRIG0(CLK := Er);
IF R_TRIG0.Q THEN TIMER := TIMER - 10; END_IF;
PANIC := PANIC;
END_PROGRAM

PROGRAM linear_congruential_generator
  VAR
    R_TRIG1 : R_TRIG;
    R_TRIG2 : R_TRIG;
    TOF0 : TOF;
    TON0 : TON;
    CTU_ULINT0 : CTU_ULINT;
    SET_TRAP : BOOL;
    Er : BOOL;
    SEED : ULINT;
    A : ULINT := 32310901;
    C : ULINT := 32310901;
    M : ULINT := 4294967296;
    M10 : ULINT := 10000;
    RANDOM_ULINT : ULINT;
    RANDOM : INT;
    D1 : INT;
    D2 : INT;
    D3 : INT;
    D4 : INT;
    RESET : BOOL;
    Clock : BOOL;
  END_VAR
  VAR  (* added by the conversion: wires and edge detectors of the diagram *)
    _MUL1_ENO : BOOL;
    _MUL1_OUT : ULINT;
    _ADD5_ENO : BOOL;
    _ADD5_OUT : ULINT;
    _MOD7_ENO : BOOL;
    _MOD7_OUT : ULINT;
    R_TRIG1_2 : R_TRIG;
  END_VAR

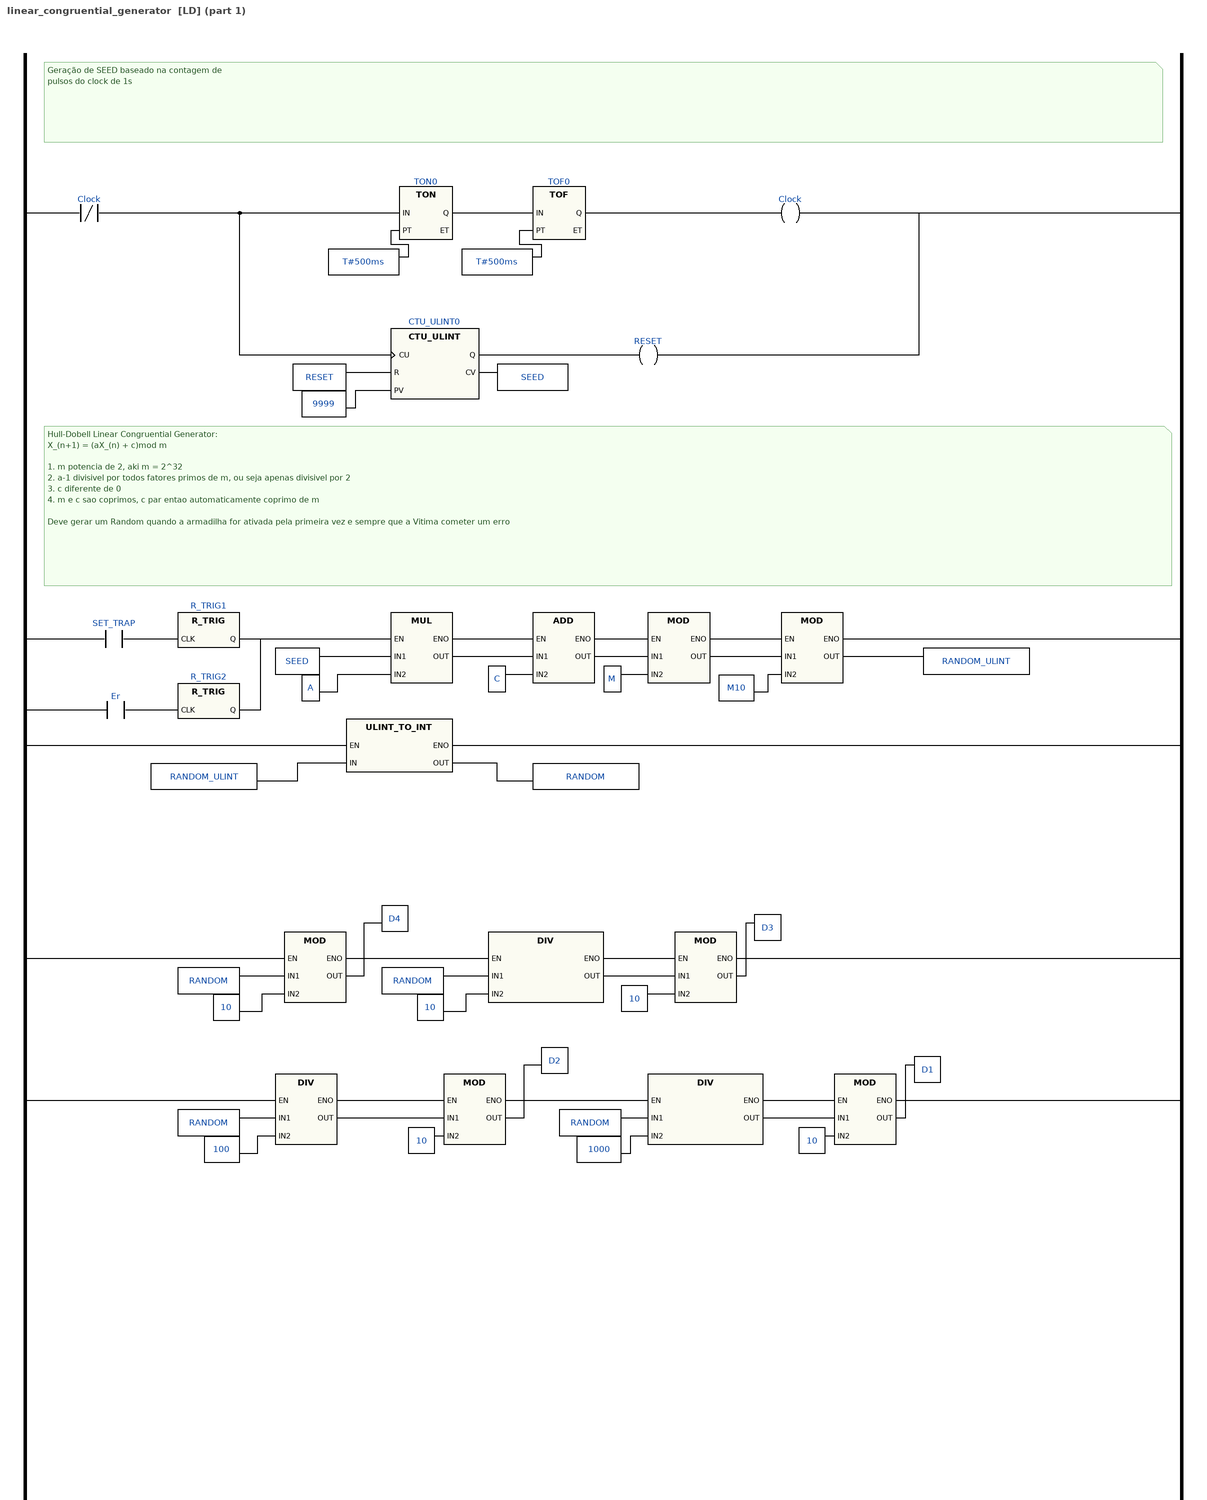
(* LD diagram, written out as Structured Text *)
(* Geração de SEED baseado na contagem de 
pulsos do clock de 1s *)
(* Hull-Dobell Linear Congruential Generator:
X_(n+1) = (aX_(n) + c)mod m

1. m potencia de 2, aki m = 2^32
2. a-1 divisivel por todos fatores primos de m, ou seja apenas divisivel por 2
3. c diferente de 0
4. m e c sao coprimos, c par entao automaticamente coprimo de m

Deve gerar um Random quando a armadilha for ativada pela primeira vez e sempre que a Vitima cometer um erro *)
R_TRIG1(CLK := SET_TRAP);
R_TRIG2(CLK := Er);
_MUL1_OUT := MUL(EN := R_TRIG1.Q OR R_TRIG2.Q, IN1 := SEED, IN2 := A, ENO => _MUL1_ENO);
_ADD5_OUT := ADD(EN := _MUL1_ENO, IN1 := _MUL1_OUT, IN2 := C, ENO => _ADD5_ENO);
_MOD7_OUT := MOD(EN := _ADD5_ENO, IN1 := _ADD5_OUT, IN2 := M, ENO => _MOD7_ENO);
IF _MOD7_ENO THEN RANDOM_ULINT := _MOD7_OUT MOD M10; END_IF;
RANDOM := ULINT_TO_INT(RANDOM_ULINT);
TON0(IN := NOT Clock, PT := T#500ms);
TOF0(IN := TON0.Q, PT := T#500ms);
Clock := TOF0.Q;
R_TRIG1_2(CLK := NOT Clock);
CTU_ULINT0(CU := R_TRIG1_2.Q, R := RESET, PV := 9999);
RESET := CTU_ULINT0.Q;
SEED := CTU_ULINT0.CV;
D4 := RANDOM MOD 10;
D3 := RANDOM / 10 MOD 10;
D2 := RANDOM / 100 MOD 10;
D1 := RANDOM / 1000 MOD 10;
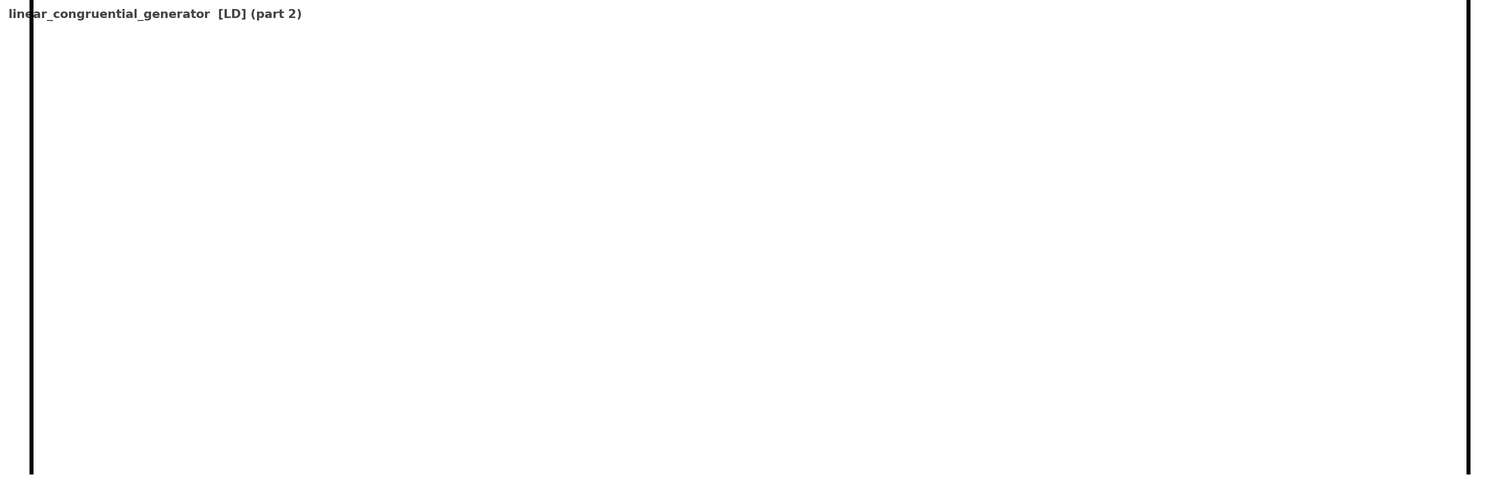
END_PROGRAM

CONFIGURATION Config0
  RESOURCE Res0 ON PLC
    TASK task0(INTERVAL := T#20ms, PRIORITY := 0);
    TASK task1(INTERVAL := T#1s, PRIORITY := 0);
    PROGRAM instance0 WITH task0 : rd_seq_rbear_trap;
    PROGRAM instance1 WITH task0 : my_clock_counter;
    PROGRAM instance2 WITH task0 : digit_extractor;
    PROGRAM instance3 WITH task0 : puzzle;
    PROGRAM instance4 WITH task0 : sub_timer;
    PROGRAM instance5 WITH task0 : linear_congruential_generator;
  END_RESOURCE
END_CONFIGURATION
